FUNCTION FC_GetMax3Arg : REAL
VAR_INPUT
	iVal1:	REAL;
	iVal2:	REAL;
	iVal3:	REAL;
END_VAR
VAR
	maxVal:	REAL;
END_VAR

maxVal := MAX(iVal1, iVal2);
maxVal := MAX(maxVal, iVal3);

FC_GetMax3Arg := maxVal;

END_FUNCTION

(* stored: Version 1.1.0.1, ProductVersion 3.1.4026.18
   POU FC_GetMax3Arg: Id {3c87efd0-572a-4abd-9e3e-313f2506644c}, SpecialFunc None *)
